Universal Robots PolyScope program: modbustest_dev.urp

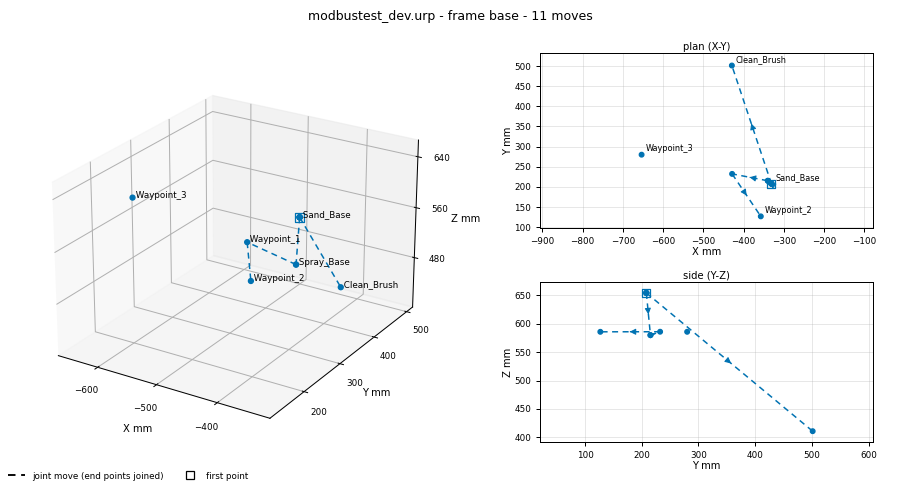
[picture p0: tool path of modbustest_dev.urp in frame base, 11 of 19 moves have a stored position in this frame; points joined in program order, loops and branches not executed]
Program modbustest_dev (installation=default directory=/programs createdIn=5.11.5.1010327 lastSavedIn=5.11.5.1010327 robotSerialNumber=20215500677)
Calibrated DH parameters: a=[0.000204, -0.239222, -0.391845, -0.000001, 0.000022, 0]; d=[0.162722, -355.808559, 353.37206, 2.570385, 0.099741, 0.099629]; alpha=[1.571124, 0.000988, 0.008295, 1.568963, -1.570303, 0]; deltaTheta=[0, -0.973091, 7.204745, 0.05153, 0, 0]
BeforeStart
  Script file /programs/cube/set_conveyor_params.script
    | def Set_Conveyor_Params(velocity, acceleration):
    | 
    |   vel_old = modbus_get_signal_status("VELOCITY_LOCAL")
    |   acc_old = modbus_get_signal_status("ACC_LOCAL")
    | 
    |   if (vel_old != velocity):
    |     modbus_set_output_register("VELOCITY_LOCAL", velocity, False)
    |     while(vel_old == modbus_get_signal_status("VELOCITY_LOCAL")):
    |       sync()
    |     end
    |     while (not(modbus_get_signal_status("VELOCITY_LOCAL")==modbus_get_signal_status("VELOCITY_REMOTE"))):
    |       sync()
    |     end
    |   end
    | 
    |   if (acc_old != acceleration):
    |     modbus_set_output_register("ACC_LOCAL", acceleration, False)
    |     while(acc_old == modbus_get_signal_status("ACC_LOCAL")):
    |       sync()
    |     end
    |     while (not(modbus_get_signal_status("ACC_LOCAL")==modbus_get_signal_status("ACC_REMOTE"))):
    |       sync()
    |     end
    |   end
    | 
    | end
  Script file /programs/cube/position_move.script
    | def Position_Move(position):
    |   mm_old = modbus_get_signal_status("MOTION_MODE_LOC")
    |   if (mm_old != position):
    |     modbus_set_output_register("MOTION_MODE_LOC",1,False)
    |     while(mm_old == modbus_get_signal_status("MOTION_MODE_LOC")):
    |       sync()
    |     end
    |     while (not(modbus_get_signal_status("MOTION_MODE_LOC")==modbus_get_signal_status("MOTION_MODE_REM"))):
    |       sync()
    |     end
    |   end
    | end
  Script file /programs/cube/distance_move.script
    | def Conveyor_Move_mm(distance):
    |   mm_old = modbus_get_signal_status("MOTION_MODE_LOC")
    |   dist_old = modbus_get_signal_status("DISTANCE_LOCAL")
    |   dir_old = modbus_get_signal_status("DIRECTION_LOCAL")
    |   id_old = modbus_get_signal_status("REQUEST_ID_LOC")
    |   if (mm_old != 0):
    |     modbus_set_output_register("MOTION_MODE_LOC",0,False)
    |     while(mm_old == modbus_get_signal_status("MOTION_MODE_LOC")):
    |       sync()
    |     end
    |     while (not(modbus_get_signal_status("MOTION_MODE_LOC")==modbus_get_signal_status("MOTION_MODE_REM"))):
    |       sync()
    |     end
    |   end
    |   distance = mm_to_steps(distance)
    |   if distance < 0:
    |     distance = distance * -1
    |     modbus_set_output_signal("DIRECTION_LOCAL", False, False)
    |   else:
    |     modbus_set_output_signal("DIRECTION_LOCAL", True, False)
    |   end
    |   if (dist_old != distance):
    |     modbus_set_output_register("DISTANCE_LOCAL",distance,False)
    |     while(dist_old == modbus_get_signal_status("DISTANCE_LOCAL")):
    |       sync()
    |     end
    |     while (not(modbus_get_signal_status("DISTANCE_LOCAL")==modbus_get_signal_status("DISTANCE_REMOTE"))):
    |       sync()
    |     end
    |   end
    |   Set_Request_Id()
    |   while(id_old == modbus_get_signal_status("REQUEST_ID_LOC")):
    |     sync()
    |   end
    |   while (not(modbus_get_signal_status("REQUEST_ID_LOC")==modbus_get_signal_status("REQUEST_ID_REM"))):
    |     sync()
    |   end
    | end
  SuppressedNode
    Script file /programs/cube/mm_move.script
      | def Conveyor_Move_mm(distance):
      |   modbus_set_output_signal("ROBOT_SENDING", True, False)
      |   modbus_set_output_register("MOTION_MODE", 0, False)
      |   distance = mm_to_steps(distance)
      |   if distance < 0:
      |   distance = distance * -1
      |   modbus_set_output_signal("DIRECTION", False, False)
      |   else:
      |   modbus_set_output_signal("DIRECTION", True, False)
      |   end
      |   modbus_set_output_register("DISTANCE", distance, False)
      |   Set_Request_Id()
      |   modbus_set_output_signal("ROBOT_SENDING", False, False)
      | end
  Script file /programs/cube/continuous_move.script
    | def Move_Continuous(direction):
    |   mm_old = modbus_get_signal_status("MOTION_MODE_LOC")
    |   if (direction == "forward"):
    |     modbus_set_output_signal("DIRECTION_LOCAL", True, False)
    |   else:
    |     modbus_set_output_signal("DIRECTION_LOCAL", False, False)
    |   end
    | if (mm_old != 2):
    |     modbus_set_output_register("MOTION_MODE_LOC",2,False)
    |     while(mm_old == modbus_get_signal_status("MOTION_MODE_LOC")):
    |       sync()
    |     end
    |     while (not(modbus_get_signal_status("MOTION_MODE_LOC")==modbus_get_signal_status("MOTION_MODE_REM"))):
    |       sync()
    |     end
    |   end
    | end
  Script file /programs/cube/idle_move.script
    | def Move_Idle():
    |   mm_old = modbus_get_signal_status("MOTION_MODE_LOC")
    |   if (mm_old != 3):
    |     modbus_set_output_register("MOTION_MODE_LOC",3,False)
    |     while(mm_old == modbus_get_signal_status("MOTION_MODE_LOC")):
    |       sync()
    |     end
    |     while (not(modbus_get_signal_status("MOTION_MODE_LOC")==modbus_get_signal_status("MOTION_MODE_REM"))):
    |       sync()
    |     end
    |   end
    | end
  Script file /programs/cube/request_id.script
    | def Set_Request_Id():
    | id = floor(random()*65000)
    | modbus_set_output_register("REQUEST_ID_LOC", id, False)
    | end
  Script file /programs/cube/steps_per_inch.script
    | def Inches_To_Steps(distance):
    | mm = distance*25.4
    | return mm_to_steps(mm)
    | end
  Script file /programs/cube/mm_to_steps.script
    | def mm_to_steps(distance):
    | teeth = 28
    | pitch = 2
    | degreesPerStep = 1.8
    | microsteps = 8
    | adjustment = 400/381
    | microStepsPerMm = 360 / teeth  / degreesPerStep / pitch * microsteps * adjustment
    | return floor(distance * microStepsPerMm)
    | end
  Script: Set_Conveyor_Params(1600, 16000)
  Script: Move_Idle()
  Script file /programs/select_job.script
    | def read_job():
    | job = modbus_get_signal_status("JOB", False)
    | #1 - cube, 2 - browser,  3 - 45
    | #4 - stereocab 2, 5 - sc 3, 6 - sc4
    | if job == 1:
    |   width = 362
    |   height = 355
    |   depth = 349
    | elif job == 2:
    |   width = 362
    |   height = 349
    |   depth = 235
    | elif job == 3:
    |   width = 724
    |   height = 235
    |   depth = 349
    | elif job == 4:
    |   width = 724
    |   height = 235
    |   depth = 349
    | elif job == 5:
    |   width = 1086
    |   height = 235
    |   depth = 349
    | elif job == 6:
    |   width = 1448
    |   height = 235
    |   depth = 349
    | elif job == 7:
    |   width = 310
    |   height = 325
    |   depth = 125
    | end
    | sleep(.2)
    | end
  loaded := 0
  dried2 := False
  Set ExpressionOutput pin=BRUSH_ON_LOCAL; expression=False
  SuppressedNode
    MoveJ speed 60 deg/s, acceleration 80 deg/s^2 (useActiveTCP=false) tcp=SandTCP; feature=Base
      Waypoint Sand_Base: TCP in base x=-331.002 y=208.013 z=654.466 mm, rx=0.0315 ry=-0.0315 rz=-1.5705 rad; joints [-61.396, -81.213, 112.495, 86.07, -50.257, -128.662] deg; TCP offset x=1.003 y=125.541 z=104.154 mm, rx=-0.7854 ry=0 rz=0 rad
Robot Program (runOnlyOnce=false)
  MoveJ speed 60 deg/s, acceleration 80 deg/s^2 (useActiveTCP=false) tcp=SandTCP; feature=Base
    Waypoint Sand_Base: TCP in base x=-331.002 y=208.013 z=654.466 mm, rx=0.0315 ry=-0.0315 rz=-1.5705 rad; joints [-61.396, -81.213, 112.495, 86.07, -50.257, -128.662] deg
  Loop While (checkContinuously=true) expression=RUN==False
    Script: read_job()
    If MOTION_MODE_LOC ≠ 3
      Script: Move_Idle()
    If FEED_CONV_LOCAL≟ True (checkContinuously=true)
      Set ExpressionOutput pin=FEED_CONV_LOCAL; expression=False
    Script: sync()
  Folder Folder
    Loop While (checkContinuously=false) expression=RUN≟ True  and JOB≟7
      Script: read_job()
      Script: Move_Continuous("forward")
      Set ExpressionOutput pin=FEED_CONV_LOCAL; expression=True
  Folder Load Workpiece
    Loop While (checkContinuously=true) expression=WORK_AT_ZERO== False  and dried2 == False and RUN == True
      If loaded≟ 0  and RUN ≟  True (checkContinuously=true)
        If MOTION_MODE_LOC != 2 (checkContinuously=true)
          Set ExpressionOutput pin=DIRECTION_LOCAL; expression=True
          Script: Move_Continuous("forward")
        Script: sync()
      If FEED_CONV_LOCAL ≟ False   and RUN ≟  True  and loaded≟ False
        Set ExpressionOutput pin=FEED_CONV_LOCAL; expression=True
        Wait DigitalInput pin=ONLOAD; digitalValue=1
        Wait DigitalInput pin=ONLOAD; digitalValue=0
        Set ExpressionOutput pin=FEED_CONV_LOCAL; expression=False
        loaded := 1
      Script: sync()
    Script: Move_Idle()
    Set ExpressionOutput pin=FEED_CONV_LOCAL; expression=False
  If RUN == True
    Script: read_job()
    Folder Sand
      MoveJ speed 60 deg/s, acceleration 80 deg/s^2 (useActiveTCP=true) feature=Base
        Waypoint Sand_Base: TCP in base x=-331.002 y=208.013 z=654.466 mm, rx=0.0315 ry=-0.0315 rz=-1.5705 rad; joints [-61.396, -81.213, 112.495, 86.07, -50.257, -128.662] deg
      MoveL speed 50 mm/s, acceleration 500 mm/s^2 (useActiveTCP=true) feature=Base
        MoveDirectionNode (selectedDirection=ZPlus toolParams=0.05, 0.5)
          Until TOOL_CONTACT_DETECTION (allowActions=false retraction=0 decelerationAcceleration=3 decelerationAngularAcceleration=34.906585)
        URCap Zero FT Sensor (Robotiq_Copilot, Robotiq Inc.) dataModel(NodeInitializedKey=true, WaitForSteadyWrenchOptionKey=true, HackTriggeringContributionIsDefinedMethodKey=true)
        URCap Finishing Tool Control (Robotiq_Copilot, Robotiq Inc.) dataModel(ToolOutputNameKey=SanderOn, HackTriggeringContributionIsDefinedMethodKey=true)
        If dried2≟ False
          Force Simple feature=Base; selection=[0, 0, 1, 0, 0, 0]; wrench=[0, 0, 6, 0, 0, 0]; limitsForce=[0.15, 0.15, 0.15, 1.047198, 1.047198, 1.047198]; limitsMotion=[0.1, 0.1, 0.1, 0.349066, 0.349066, 0.349066]
            Script: Conveyor_Move_mm(width-12)
            Wait Condition expression=SERVER_STATE==1
            Folder moveHeight
              currentPosition := get_actual_tcp_pose()
              newPosition := pose_add(currentPosition, p[-height/1000,0,0,0,0,0])
              Waypoint Waypoint (Variable): variable=newPosition
            Script: Conveyor_Move_mm(-width+12)
            Wait Condition expression=SERVER_STATE==1
            Folder moveHeight
              currentPosition := get_actual_tcp_pose()
              newPosition := pose_add(currentPosition, p[height/1000,0,0,0,0,0])
              Waypoint Waypoint (Variable): variable=newPosition
            URCap Finishing Tool Control (Robotiq_Copilot, Robotiq Inc.) dataModel(FinishingToolStateKey=false, ToolOutputNameKey=SanderOn, HackTriggeringContributionIsDefinedMethodKey=true)
        Else 
          Force Simple feature=Base; selection=[0, 0, 1, 0, 0, 0]; wrench=[0, 0, 6, 0, 0, 0]; limitsForce=[0.15, 0.15, 0.15, 1.047198, 1.047198, 1.047198]; limitsMotion=[0.1, 0.1, 0.1, 0.349066, 0.349066, 0.349066]
            Script: Conveyor_Move_mm(width-12)
            Wait Condition expression=SERVER_STATE==1
            Folder moveHeight
              currentPosition := get_actual_tcp_pose()
              newPosition := pose_add(currentPosition, p[-height/1000,0,0,0,0,0])
              Waypoint Waypoint (Variable): variable=newPosition
            Script: Conveyor_Move_mm(-width+12)
            Wait Condition expression=SERVER_STATE==1
            Folder moveHeight
              currentPosition := get_actual_tcp_pose()
              newPosition := pose_add(currentPosition, p[height/1000,0,0,0,0,0])
              Waypoint Waypoint (Variable): variable=newPosition
            URCap Finishing Tool Control (Robotiq_Copilot, Robotiq Inc.) dataModel(FinishingToolStateKey=false, ToolOutputNameKey=SanderOn, HackTriggeringContributionIsDefinedMethodKey=true)
      MoveJ speed 60 deg/s, acceleration 80 deg/s^2 (useActiveTCP=true) feature=Base
        Waypoint Sand_Base: TCP in base x=-331.002 y=208.013 z=654.466 mm, rx=0.0315 ry=-0.0315 rz=-1.5705 rad; joints [-61.396, -81.213, 112.495, 86.07, -50.257, -128.662] deg
    Folder 45 Sand [hidden by the author, left out]
    Folder SC 3 and 4 Sand [hidden by the author, left out]
    Folder Spray Vertical
      MoveJ speed 60 deg/s, acceleration 80 deg/s^2 (useActiveTCP=false) tcp=SprayTCP; feature=Base
        Waypoint Spray_Base: TCP in base x=-340.005 y=215.234 z=580.009 mm, rx=0.0001 ry=-0.0001 rz=0.0032 rad; joints [-52.421, -78.551, 119.412, 80.396, -56.251, 42.834] deg; TCP offset x=63.143 y=-107.882 z=84.395 mm, rx=0.6139 ry=0.6139 rz=-1.4822 rad
        If JOB == 2
          MoveL speed 250 mm/s, acceleration 1200 mm/s^2 (useActiveTCP=true) feature=Base
            MoveDirectionNode (selectedDirection=ZPlus)
              Until DISTANCE (allowActions=false deceleration=3 distanceNodeType=STOP) Distance=0.1; motionParameters(blendRadius=0)
        If JOB == 7
          MoveL speed 250 mm/s, acceleration 1200 mm/s^2 (useActiveTCP=true) feature=Base
            MoveDirectionNode (selectedDirection=ZPlus)
              Until DISTANCE (allowActions=false deceleration=3 distanceNodeType=STOP) Distance=0.2; motionParameters(blendRadius=0)
        Set DigitalOutput pin=digital_out[5]; digitalValue=1
      MoveL speed 50 mm/s, acceleration 500 mm/s^2 (useActiveTCP=true) feature=Base
        Script: Conveyor_Move_mm(width-12)
        Wait Condition expression=SERVER_STATE==1
        Folder moveHeight
          currentPosition := get_actual_tcp_pose()
          newPosition := pose_add(currentPosition, p[-height/1000,0,0,0,0,0])
          Waypoint Waypoint (Variable): variable=newPosition
        Script: Conveyor_Move_mm(-width+12)
        Wait Condition expression=SERVER_STATE==1
        Folder moveHeight
          currentPosition := get_actual_tcp_pose()
          newPosition := pose_add(currentPosition, p[height/1000,0,0,0,0,0])
          Waypoint Waypoint (Variable): variable=newPosition
          Set DigitalOutput pin=digital_out[5]; digitalValue=0
      MoveJ speed 60 deg/s, acceleration 80 deg/s^2 (useActiveTCP=true) feature=Base
        Waypoint Spray_Base: TCP in base x=-340.005 y=215.234 z=580.009 mm, rx=0.0001 ry=-0.0001 rz=0.0032 rad; joints [-52.421, -78.551, 119.412, 80.396, -56.251, 42.834] deg
    Folder 45 Spray [hidden by the author, left out]
    Folder SC 3 and 4 Spray [hidden by the author, left out]
    Folder Cube
      If JOB==1
        Folder Spray Horizontal
          MoveJ speed 60 deg/s, acceleration 80 deg/s^2 (useActiveTCP=false) tcp=SprayTCP; feature=Base
            Waypoint Waypoint_1: TCP in base x=-428.6 y=232.291 z=586.04 mm, rx=0.0002 ry=0.7854 rz=-0.0001 rad; joints [-31.287, -77.017, 103.348, -116.368, 90.409, -148.974] deg
            Set DigitalOutput pin=digital_out[5]; digitalValue=1
            Script: Conveyor_Move_mm(width-12)
            Wait Condition expression=SERVER_STATE==1
            Set DigitalOutput pin=digital_out[5]; digitalValue=0
            Waypoint Waypoint_2: TCP in base x=-357.369 y=126.847 z=585.919 mm, rx=-0.6139 ry=0.6139 rz=1.4822 rad; joints [-30.772, -119.042, 138.633, -109.626, 90.417, -59.463] deg
            MoveL speed 50 mm/s, acceleration 500 mm/s^2 (useActiveTCP=true) feature=Base
              Set DigitalOutput pin=digital_out[5]; digitalValue=1
              Folder moveHeight
                currentPosition := get_actual_tcp_pose()
                newPosition := pose_add(currentPosition, p[-height/1000,0,0,0,0,0])
                Waypoint Waypoint (Variable): variable=newPosition
              Set DigitalOutput pin=digital_out[5]; digitalValue=0
            Script: Conveyor_Move_mm(-width+12)
            Waypoint Waypoint_3: TCP in base x=-653.365 y=279.996 z=585.94 mm, rx=0.6141 ry=0.6138 rz=-1.4822 rad; joints [-37.861, -42.297, 48.999, -96.723, 90.48, 127.774] deg
            Wait Condition expression=SERVER_STATE==1
            MoveL speed 50 mm/s, acceleration 500 mm/s^2 (useActiveTCP=true) feature=Base
              Set DigitalOutput pin=digital_out[5]; digitalValue=1
              Folder moveHeight
                currentPosition := get_actual_tcp_pose()
                newPosition := pose_add(currentPosition, p[height/1000,0,0,0,0,0])
                Waypoint Waypoint (Variable): variable=newPosition
              Set DigitalOutput pin=digital_out[5]; digitalValue=0
    MoveJ speed 60 deg/s, acceleration 80 deg/s^2 (useActiveTCP=false) tcp=SandTCP; feature=Base
      Waypoint Sand_Base: TCP in base x=-331.002 y=208.013 z=654.466 mm, rx=0.0315 ry=-0.0315 rz=-1.5705 rad; joints [-61.396, -81.213, 112.495, 86.07, -50.257, -128.662] deg; TCP offset x=1.003 y=125.541 z=104.154 mm, rx=-0.7854 ry=0 rz=0 rad
    Folder Clean Spray
      MoveJ speed 60 deg/s, acceleration 80 deg/s^2 (useActiveTCP=false) tcp=SandTCP; feature=Base
        Waypoint Sand_Base: TCP in base x=-331.002 y=208.013 z=654.466 mm, rx=0.0315 ry=-0.0315 rz=-1.5705 rad; joints [-61.396, -81.213, 112.495, 86.07, -50.257, -128.662] deg
        Waypoint Clean_Brush: TCP in base x=-429.199 y=501.374 z=410.614 mm, rx=-1.4653 ry=-0.4723 rz=0.6515 rad; joints [-67.004, -62.545, 104.831, 88.525, -82.288, -342.283] deg
        MoveL speed 50 mm/s, acceleration 500 mm/s^2 (useActiveTCP=true) feature=Base
          MoveDirectionNode (selectedDirection=ZPlus)
            Until TOOL_CONTACT_DETECTION (allowActions=false retraction=0.003)
        Wait Sleep waitTime=1
        Set ExpressionOutput pin=BRUSH_ON_LOCAL; expression=True
        Timer (action=Start) variable(name=timer_brush)
    If dried2≟ False
      Folder Dry
        Timer (action=Start) variable(name=timer_dry)
        Script: Conveyor_Move_mm(width+500)
        Wait Condition expression=SERVER_STATE==1
        Loop While (checkContinuously=false) expression=timer_dry<165
          Script: Conveyor_Move_mm(-(width/2))
          Wait Condition expression=SERVER_STATE==1
          Script: Conveyor_Move_mm(width/2)
          Wait Condition expression=SERVER_STATE==1
        Script: Move_Continuous("reverse")
        Wait DigitalInput pin=WORK_AT_ZERO; digitalValue=1
        Wait DigitalInput pin=WORK_AT_ZERO; digitalValue=0
        Script: Move_Continuous("forward")
        Wait DigitalInput pin=WORK_AT_ZERO; digitalValue=1
        dried2 := True
        Timer (action=Stop) variable=timer_dry
        Timer (action=Reset) variable=timer_dry
        Script: Move_Idle()
    Else 
      Folder Folder
        Loop While (checkContinuously=false) expression=OFFLOAD≠ False
          Script: Move_Continuous("forward")
  SuppressedNode
    Folder Motion Test
      Wait Sleep waitTime=1
      Script: Conveyor_Move_mm(width)
      Wait Condition expression=SERVER_STATE == 1
      Script: Conveyor_Move_mm(-width)
      Wait Condition expression=SERVER_STATE == 1
  Script: sync()
Thread Thread_1 (runOnlyOnce=false)
  If RUN == False (checkContinuously=true)
    If MOTION_MODE_LOC ≠3 (checkContinuously=true)
      Script: Move_Idle()
    If FEED_CONV_LOCAL≟ True (checkContinuously=true)
      Set ExpressionOutput pin=FEED_CONV_LOCAL; expression=False
    Script: sync()
  Else 
    Script: sync()
Thread Thread_2 (runOnlyOnce=false)
  If timer_brush > 30 (checkContinuously=true)
    Set ExpressionOutput pin=BRUSH_ON_LOCAL; expression=False
    Wait Sleep waitTime=1
    Timer (action=Stop) variable=timer_brush
    Timer (action=Reset) variable=timer_brush
    SuppressedNode
      If dried≟ False
        MoveL speed 250 mm/s, acceleration 1200 mm/s^2 (useActiveTCP=true) feature=Base
          MoveDirectionNode (selectedDirection=ZMinus)
            Until DISTANCE (allowActions=false deceleration=3 distanceNodeType=STOP) Distance=0.02; motionParameters(blendRadius=0)
  Script: sync()
